ABB RobotStudio station: SC Infeeder finished.rspag

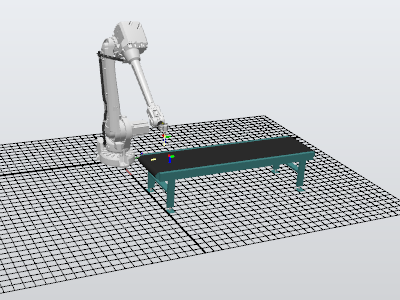
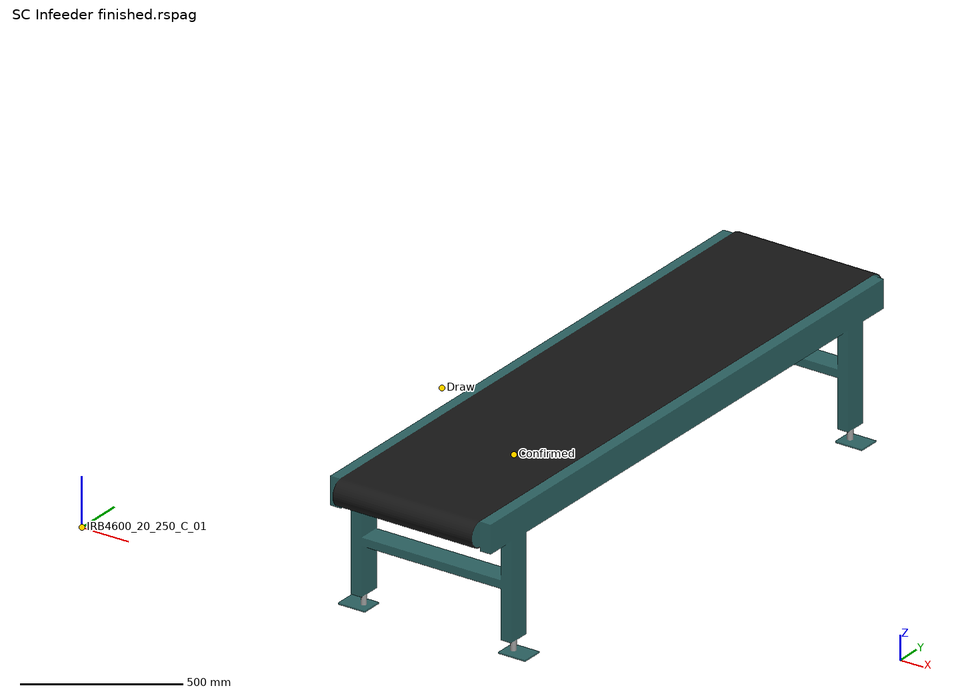
[picture v1: parts stored in the station drawn from their meshes, with robot base, taught points and paths (robot models come from the ABB library and are not in the file)]
--- station ---
Station SC Infeeder finished (saved by RobotStudio 23.4.10609.1)
Controller IRB4600
  mechanical unit ROB_1: IRB4600_20_250_C_01, 6 joints, base frame (0, 0, 0) mm
Layout (positions relative to the parent item):
  - IRB4600_20_250_C_01 [mechanism, from %ABB.RobotStudio.Models.IRB4600%\IRB4600_20_250_C_G_01.rslib] at (0, 0, 0) mm; joint values [0.065, -0.1396, 0.8384, 0.1009, -0.7014, -0.0772] (rad or m)
  - Belt Conveyor [part], size 703.5 x 2188.6 x 501 mm
  - Box [part], size 500 x 300 x 200 mm
  - SC_InFeeder [smart component]
      signals: DO doBoxInPos, DI diPauseConveyor, DO doConveyorPaused
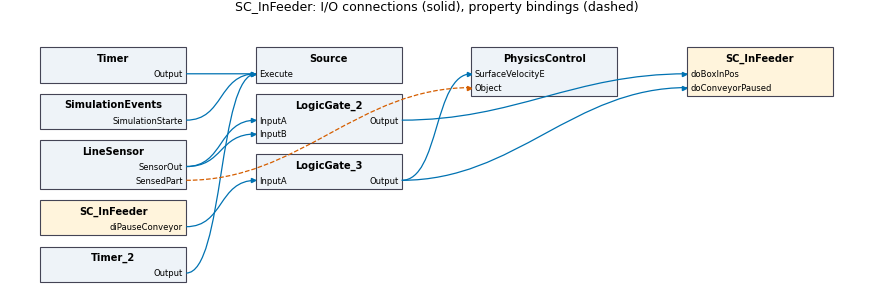
      connections:
        Timer.Output -> Source.Execute
        SimulationEvents.SimulationStarted -> Source.Execute
        LineSensor.SensorOut -> LogicGate_2.InputA
        LineSensor.SensorOut -> LogicGate_2.InputB
        LogicGate_2.Output -> SC_InFeeder.doBoxInPos
        SC_InFeeder.diPauseConveyor -> LogicGate_3.InputA
        LogicGate_3.Output -> PhysicsControl.SurfaceVelocityEnabled
        LogicGate_3.Output -> SC_InFeeder.doConveyorPaused
        Timer_2.Output -> Source.Execute
        LineSensor.SensedPart => PhysicsControl.Object
    - Source [smart component, from Components\Source.rslib]
        properties: Source=Box; Copy=(none); Parent=(none); Position=[0 0 0]; Orientation=[0 0 0]; Transient=true; PhysicsBehavior=3
    - LineSensor [smart component, from Components\LineSensor.rslib]
        properties: Start=[1.3 -0.09 0.547]; End=[1.3 -0.03 0.547]; Radius=0; SensedPart=(none); SensedPoint=[0 0 0]; Length=0.06; Tag=(none)
      - _sensorPart_ [part], size 0 x 60 x 0 mm
    - LogicGate_2 [smart component, from Components\LogicGate.rslib]
        properties: Operator=OR; Delay=0
    - SimulationEvents [smart component, from Components\SimulationEvents.rslib]
    - PhysicsControl [smart component, from Components\PhysicsControl.rslib]
        properties: Object=(none); Behavior=3; SurfaceVelocity=0
    - LogicGate_3 [smart component, from Components\LogicGate.rslib]
        properties: Operator=NOT; Delay=0
    - Timer_2 [smart component, from Components\Timer.rslib]
        properties: StartTime=0; Interval=5; Repeat=true; CurrentTime=12.984
  - Belt [part], size 529.1 x 2200.3 x 102.1 mm
  - Pen [mechanism, from Training Objects\Pen.rslib] at (1160.02, 70, 921.71) mm, rotated rx 0 ry 90 rz 0 deg
  - SC_Painter [smart component] at (1300.02, 70, 811.71) mm
      connections:
        LineSensor.SensorOut -> PaintApplicator_4.Enabled
        LineSensor.SensedPart => PaintApplicator_4.Part
    - PaintApplicator_4 [smart component, from Components\PaintApplicator.rslib] at (0, 0, -81.83) mm
        properties: Part=(none); Color=-16744256; ShowPreviewCone=true; Strength=0.5; Range=0.5; Width=0.5; Height=0.5
    - LineSensor [smart component, from Components\LineSensor.rslib]
        properties: Start=[2.81766896481628E-08 -8.9564643340756E-09 -0.111707072267828]; End=[0 0 0.1]; Length=0.21170707226783; Radius=0; Tag=(none); SensedPart=pen; SensedPoint=[1.30002294921875 0.07 0.81170703125]
      - _sensorPart_ [part], size 0 x 0 x 211.7 mm
Attachment: Pen is attached to IRB4600_20_250_C_01 / Link6
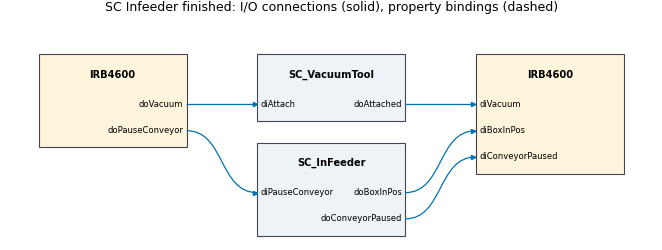
Station logic (signal -> signal, property => property):
  SC_VacuumTool.doAttached -> IRB4600.diVacuum
  IRB4600.doVacuum -> SC_VacuumTool.diAttach
  SC_InFeeder.doBoxInPos -> IRB4600.diBoxInPos
  SC_InFeeder.doConveyorPaused -> IRB4600.diConveyorPaused
  IRB4600.doPauseConveyor -> SC_InFeeder.diPauseConveyor

--- Backups/IRB4600/RAPID/TASK1/PROGMOD/CalibData.mod ---
MODULE CalibData
	PERS tooldata tVacuum:=[TRUE,[[0,0,150],[1,0,0,0]],[9,[0,0,100],[1,0,0,0],0,0,0]];
	TASK PERS wobjdata wobjInFeeder:=[FALSE,TRUE,"",[[0,0,0],[1,0,0,0]],[[1000,-80,497],[1,0,0,0]]];
    PERS tooldata Pen_TCP:=[TRUE,[[110,0,140],[0.707106781,0,0.707106781,0]],[1,[10.7435139,0,140],[1,0,0,0],0,0,0]];
ENDMODULE

--- Backups/IRB4600/RAPID/TASK1/PROGMOD/Module1.mod ---
MODULE Module1
    CONST robtarget pPick:=[[300.023,150,209.481],[0,-0.707106781,0.707106781,0],[0,0,0,0],[9E+09,9E+09,9E+09,9E+09,9E+09,9E+09]];
    CONST robtarget Draw:=[[300.022993432,150.000002947,314.707147681],[0.000000011,0,1,0],[0,0,-1,1],[9E+09,9E+09,9E+09,9E+09,9E+09,9E+09]];
    CONST robtarget Confirmed:=[[616.591587907,80,203.883134],[-0.000000001,0,1,0],[0,0,0,0],[9E+09,9E+09,9E+09,9E+09,9E+09,9E+09]];
    !***********************************************************
    !
    ! Module:  Module1
    !
    ! Description:
    !   <Insert description here>
    !
    ! Author: ander
    !
    ! Version: 1.0
    !
    !***********************************************************


    !***********************************************************
    !
    ! Procedure main
    !
    !   Smart Component example, Pick and Place application.

    !
    !***********************************************************
    PROC main()
        WHILE TRUE DO
            PickPart;
        ENDWHILE
    ENDPROC

    PROC PickPart()
        !** The robot moves to a wait position 200 mm above the pick position. **
        !** The robot waits for a box to pick at the infeeder stop. **
        !** The robot goes to the pick position. **
        !** To attach the box, the robot turns on the digital output signal "doVacuum" which is connected to the Smart Component "SC_VacuumTool". **
        !** The robot waits for the digital input signal "diVacuum" to goes high, which comes from "SC_VacuumTool" and indicates that the box is attached. **
        !** The robot moves up from the infeeder. **
        !** The robot moves to the drop position above the pallet. **
        !** To detach the box, the robot turns off the digital output signal "doVacuum" which is connected to the Smart Component "SC_VacuumTool". **
        !** The robot waits for the digital input signal "diVacuum" to goes low, which comes from "SC_VacuumTool" and indicates that the box is detached. **
        !** The wait time simulates the time it takes for a real vacuum gripper to loose the vacuum. **
        MoveJ Draw,v300,fine,Pen_TCP\WObj:=wobjInFeeder;
    ENDPROC
    PROC Path_10()
        MoveL Confirmed,v300,fine,Pen_TCP\WObj:=wobjInFeeder;
    ENDPROC
ENDMODULE

--- Backups/IRB4600/SYSPAR/EIO.cfg ---
EIO:CFG_1.0:6:1::
#
EIO_SIGNAL:

      -Name "doVacuum" -SignalType "DO" -Access "All"

      -Name "diVacuum" -SignalType "DI" -Access "All"

      -Name "diBoxInPos" -SignalType "DI" -Access "All"

      -Name "doPauseConveyor" -SignalType "DO" -Access "All"

      -Name "diConveyorPaused" -SignalType "DI" -Access "All"
